{attribute 'Tc2GvlVarNames'}
{attribute 'strict'}
//Tipologia di WorkArea
TYPE e_Tipo_WorkArea :
(
	TYPOLOGY_NOT_DEFINED		:= -1,	(* Tipologia NON Definita *)			
	TYPOLOGY_STACK				:= 1,	(* Tipologia Catasta Vuoti *)
	TYPOLOGY_PALLET				:= 2,	(* Tipologia Postazione Di Lavoro in WorkArea *)
	TYPOLOGY_LAYER				:= 3,	(* Tipologia Postazione Magazzino Falde in WorkArea *)
	
	TYPOLOGY_OVER_TRANSPORT		:= 5,   (* Tipologia Di Postazione di prelievo/deposito su trasporti (rulliere o catenaria) *)
	TYPOLOGY_BUNDLE				:= 6,   (* Tipologia Di Postazione Di deposito = BUNDLE *)
	TYPOLOGY_ALIGNER			:= 7,   (* Tipologia Di Postazione Di PAREGGIATURA *)
	
	TYPOLOGY_WASTE				:= 8,	(* Tipologia Di Postazione SCARTI *)

	
	TYPOLOGY_EXTERNAL_DEPPREL	:= 10(* Tipologia Postazione ESTERNA al perimetro del Pallettizzatore: Utilizzata per deposito o prelievo di Pallet/Casse/Cavalline lavorate o da lavorare *)
);
END_TYPE
//  TYPOLOGY_NOT_DEFINED = '-1'

(* stored: Version 1.1.0.1, ProductVersion 3.1.4024.11
   EnumerationTextList e_Tipo_WorkArea: Id {58222ab8-16ab-4a2a-86d8-896c9107c267} *)
